PROGRAM PRG_QueueTest
VAR
	stQueue : ST_Queue;
	fbQueue : FB_Queue;
	
	bInit : BOOL := FALSE;
	iResult : DINT;
	bResult : BOOL;
	
END_VAR


	fbQueue.Enqueue(1);
	fbQueue.Enqueue(2);
	fbQueue.Enqueue(3);
	fbQueue.Enqueue(4);
	fbQueue.Enqueue(5);
	fbQueue.Enqueue(6);
	fbQueue.Enqueue(7);
	fbQueue.Enqueue(8);
	fbQueue.Enqueue(9);
	fbQueue.Enqueue(10);
	fbQueue.Enqueue(11);
	iResult := fbQueue.Dequeue(); // 1
	iResult := fbQueue.Dequeue();
	iResult := fbQueue.Dequeue();
	iResult := fbQueue.Dequeue();
	iResult := fbQueue.Dequeue(); // 5
	iResult := fbQueue.Dequeue();
	iResult := fbQueue.Dequeue();
	iResult := fbQueue.Dequeue();
	iResult := fbQueue.Dequeue();
	iResult := fbQueue.Dequeue(); // 10
	iResult := fbQueue.Dequeue(); // element 11; should fail

END_PROGRAM

(* stored: Version 1.1.0.1, ProductVersion 3.1.4024.6
   POU PRG_QueueTest: Id {178e8df6-feea-4e4a-b787-9319e10c1557}, SpecialFunc None *)
